FUNCTION_BLOCK EHWCheckValid
VAR_INPUT
	rBarcodeReading : REAL;  	// current barcode reading
	tsTrack : ST_Track_Segment_EHC; 	// current track segment
END_VAR
VAR_OUTPUT
	bResult : BOOL;
END_VAR
VAR
END_VAR

bResult := FALSE;

IF tsTrack.rStart < tsTrack.rEnd THEN
	IF rBarcodeReading >= tsTrack.rStart + 0.2 AND rBarcodeReading <= tsTrack.rEnd - 0.2 THEN
		bResult := TRUE;
	END_IF
ELSE
	IF rBarcodeReading <= tsTrack.rStart - 0.2 AND rBarcodeReading >= tsTrack.rEnd + 0.2 THEN
		bResult := TRUE;
	END_IF
END_IF

END_FUNCTION_BLOCK

(* stored: Version 1.1.0.1
   POU EHWCheckValid: Id {254c733d-6fa6-4074-b39e-0df2fec2ab4c}, SpecialFunc None *)
